# EPICS StreamDevice protocol: mks937bApp/protocol/mks937b.protocol
# Stream Device Protocol for the MKS 937B Multi-Sensor System
# This protocol uses features defined in Stream Device Version 2
#
# Ian Gillingham - April 2010
#
# $1 = address, Controller address (001 .. 253)
# $2 = channel number: 1 - 5
# $3 = setpoint: 1 - 12

locktimeout = 5000;
terminator   = ";FF";
replytimeout = 1000;
readtimeout  = 1000;
extrainput   = Ignore;

# The 937B appears to have preamble on all commands and responses
# of the form '@<aaa>', where aaa is the unit number (1-254)
# presumably to cater for multidrop RS485 for multiple controllers.
# Default here to assume just one unit (as on RS232). Will need to make this variable if RS485 is ever implemented.
unitid = 1;

# Send an initial dummy command to clear out any garbage the mks has already received.
# This makes it more likely that the first command sent is received OK.
# NB we dont wait for a response to the dummy command because if it didnt arrive (e.g. rs232 unplugged) then
# streams would issue a replyTimeout exception and stop the ioc.
@init{out " ";}

pressure { out "@\$1PR\$2?"; in "\$1ACK%f"; @mismatch{} }
raw      { out "@\$1PR\$2?"; in "\$1ACK%s"; }
status   { out "@\$1PR\$2?"; in "\$1ACK%{\?.|  \?E|OVER|ATM|<1.00E-11|RF_OFF|OFF|WAIT|L|CTRL_OFF|PROT_OFF|NOGAUGE|MISCONN|NOT|Not|C}"; }
ccenable { out "@\$1%{CP\$2!OFF|CP\$2!ON}"; in "\$1ACK%{OFF|ON}"; }
get_cc_enabled{ out "@\$1CP\$2?"; in "\$1ACK%{OFF|ON}"; }
pirgenable { out "@\$1%{CP\$2!OFF|CP\$2!ON}"; in "\$1ACK%{OFF|ON}"; }
get_gauge_enabled { out "@\$1CP\$2?"; in "\$1ACK%{OFF|ON}"; }

# Relay setpoints
getsp   { out "@\$1SP\$2?"; in "\$1ACK%f"; }
setsp   { out "@\$1SP\$2!%0.1E"; in "\$1ACK"; }
dissp   { out "@\$1\$2!0"; in "\$1ACK"; }

# Relay Hysteresis
getrelay_hyst   { out "@\$1SH\$2?"; in "\$1ACK%f"; }
setrelay_hyst   { out "@\$1SH\$2!%0.1E"; in "\$1ACK"; }

# Relay mode
getrelay_mode   { out "@\$1EN\$2?"; in "\$1ACK%{SET|CLEAR|ENABLE}"; }
setrelay_mode   { out "@\$1EN\$2!%{SET|CLEAR|ENABLE}"; in "\$1ACK"; }

# Relay direction
getrelay_direction   { out "@\$1SD\$2?"; in "\$1ACK%{ABOVE|BELOW}"; }
setrelay_direction   { out "@\$1SD\$2!%{ABOVE|BELOW}"; in "\$1ACK"; }

# Protection (overpressure) setpoints
getpro   { out "@\$1PRO\$2?"; in "\$1ACK%f"; }
setpro   { out "@\$1PRO\$2!%0.1E"; in "\$1ACK"; }
dispro   { out "@\$1PRO\$2!0"; in "\$1ACK"; }

# TTL trigger setpoints
getfrc_sp  { out "@\$1FRC\$2?"; in "\$1ACK%f"; }
setfrc_sp  { out "@\$1FRC\$2!%0.1E"; in "\$1ACK"; }

# CC control
getcc_sp   { out "@\$1CSP\$2?"; in "\$1ACK%f"; }
setcc_sp   { out "@\$1CSP\$2!%0.1E"; in "\$1ACK"; }
discc_sp   { out "@\$1CSP\$2!%0.1E"; in "\$1ACK"; }
getcc_hyst { out "@\$1CHP\$2?"; in "\$1ACK%f"; }
setcc_hyst { out "@\$1CHP\$2!%0.1E"; in "\$1ACK"; }
getcc_ctl  { out "@\$1CTL\$2?"; in "\$1ACK%{OFF|SAFE|AUTO}"; }
setcc_ctl  { out "@\$1CTL\$2!%{OFF|SAFE|AUTO}"; in "\$1ACK"; }
getcc_ctrl_chan  { out "@\$1CSE\$2?"; in "\$1ACK%{C1|C2|OFF|A1|B1|A2|B2}"; }
setcc_ctrl_chan  { out "@\$1CSE\$2!%{C1|C2|OFF|A1|B1|A2|B2}"; in "\$1ACK"; }

# Controller parameters

unit    { out "@\$1U?"; in "\$1ACK%s"; }
ctlv    { out "@\$1FV6?"; in "\$1ACK%f"; }
comv    { out "@\$1FV5?"; in "\$1ACK%f";  @mismatch{};}
modcc   { out "@\$1MT?"; in "\$1ACK%{HC|CC|PR|CV|TC|CM|P1|C1|T1|M1|NC|WC}"; }
moda    { out "@\$1MT?"; in "\$1ACK\?\?,%{HC|CC|PR|CV|TC|CM|P1|C1|T1|M1|NC|WC}"; }
modb    { out "@\$1MT?"; in "\$1ACK\?\?,\?\?,%{HC|CC|PR|CV|TC|CM|P1|C1|T1|M1|NC|WC}"; }

#debug
debug { ExtraInput = Ignore; out "%s"; in "%s"}
